// TIA Portal V17 export
// export: Created 2022-07-16T16:56:10.9456586Z, ExportSetting WithDefaults, DisplayName Totally Integrated Automation Portal, DisplayVersion V17, DisplayName TIA Portal Openness, DisplayVersion V17, DisplayName TIA Portal Version Control Interface, DisplayVersion V17, DisplayName TIA Portal Test Suite Advanced, DisplayVersion V17, DisplayName STEP 7 Professional, DisplayVersion V17, DisplayName STEP 7 Safety, DisplayVersion V17, DisplayName WinCC Professional, DisplayVersion V17
TYPE "readWriteListType"
// stored: IsFailsafeCompliant false
   STRUCT
      NodeCount { ExternalAccessible := 'False'; ExternalVisible := 'False'; ExternalWritable := 'False'} : UInt;
      Nodes { ExternalAccessible := 'False'; ExternalVisible := 'False'; ExternalWritable := 'False'; S7_SetPoint := 'True'} : Array[0.."READ_LIST_COUNT"] of OPC_UA_NodeId;
      NodeHdls { ExternalAccessible := 'False'; ExternalVisible := 'False'; ExternalWritable := 'False'} : Array[0.."READ_LIST_COUNT"] of DWord;
   END_STRUCT;
   // Nodes[0..2].NamespaceIndex := 0;
   // Nodes[0].Identifier := WSTRING#'"OPC_UA_Interface"."startCounting"';
   // Nodes[1].Identifier := WSTRING#'"OPC_UA_Interface"."actValue"';
   // Nodes[2].Identifier := WSTRING#'"OPC_UA_Interface"."endValue"';
   // Nodes[0..2].IdentifierType := 1;
END_TYPE
